(* CoDeSys 2.3.9.13 project: Stepper_03_Example01.pro *)
(* Libraries: D:\Daten\CodeSys_841\Projekte\Stepper\MC3\Release0.9.6\Stepper_03.lib 7.10.09 08:41:07, Standard.lib 22.11.04 11:21:12 *)

(* PLC configuration (modules and I/O channels)
Module Fieldbus Assignment [WAGO_Module] node 0, in %IB0 out %QB0 {INTTypePAAssignment = PLC; INTTypeModule = plugged}
Module Fieldbus Assignment [WAGO_Module] node 1, in %IB1 out %QB1 {INTTypePAAssignment = PLC; INTTypeModule = plugged}
Fieldbus variables [FB_VARS] node 1, in %IB0 out %QB0
*)

(* POU PLC_PRG, FBD *)
PROGRAM PLC_PRG
VAR
	Stepper_673					: MC3_StepperCommunication;
	Stepper1						: MC3_StepperVisu:=(	BasicModule:=673);

	Stepper1In 	AT%IB0		: ARRAY[0..11] OF BYTE;		(* input address stepper modul 750-673 *)
	Stepper1Out  	AT%QB0 		: ARRAY[0..11] OF BYTE;		(* output address stepper modul 750-673 *)


	startablauf						: BOOL;
	ablaufstate					: INT;
	error							: BOOL;
	count							: INT;
	testcount						: INT;
	TON1							: TON;
END_VAR
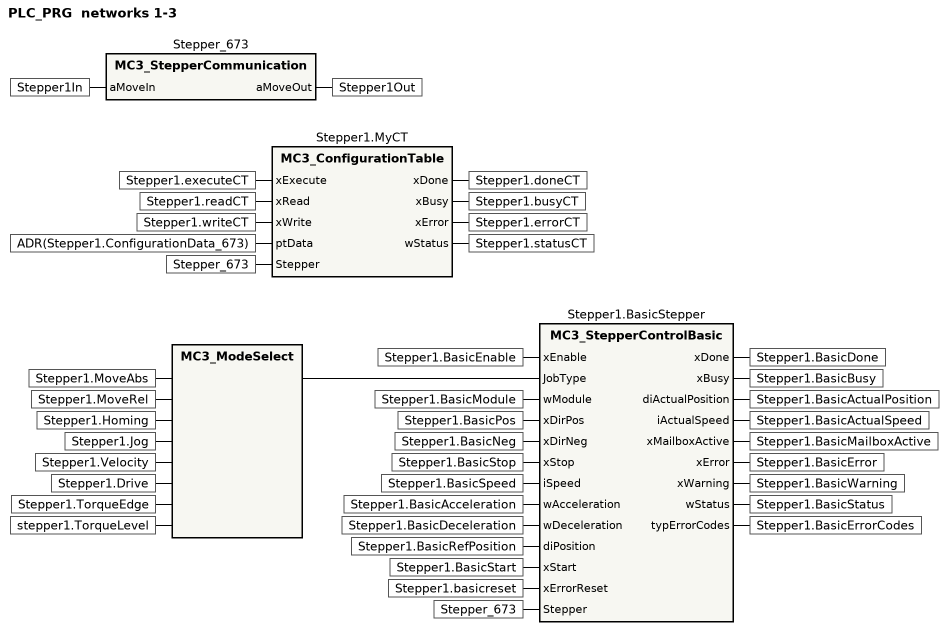
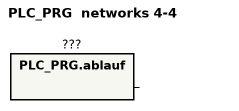
_FBD_ (* Function Block Diagram *)
NETWORK 1
	Stepper_673:MC3_StepperCommunication(aMoveIn: Stepper1In) => Stepper1Out
NETWORK 2
	Stepper1.MyCT:MC3_ConfigurationTable(xExecute: Stepper1.executeCT, xRead: Stepper1.readCT, xWrite: Stepper1.writeCT, ptData: ADR(Stepper1.ConfigurationData_673), Stepper: Stepper_673, xBusy => Stepper1.busyCT, xError => Stepper1.errorCT, wStatus => Stepper1.statusCT) => Stepper1.doneCT
NETWORK 3
	Stepper1.BasicStepper:MC3_StepperControlBasic(xEnable: Stepper1.BasicEnable, JobType: MC3_ModeSelect(Stepper1.MoveAbs, Stepper1.MoveRel, Stepper1.Homing, Stepper1.Jog, Stepper1.Velocity, Stepper1.Drive, Stepper1.TorqueEdge, stepper1.TorqueLevel), wModule: Stepper1.BasicModule, xDirPos: Stepper1.BasicPos, xDirNeg: Stepper1.BasicNeg, xStop: Stepper1.BasicStop, iSpeed: Stepper1.BasicSpeed, wAcceleration: Stepper1.BasicAcceleration, wDeceleration: Stepper1.BasicDeceleration, diPosition: Stepper1.BasicRefPosition, xStart: Stepper1.BasicStart, xErrorReset: Stepper1.basicreset, Stepper: Stepper_673, xBusy => Stepper1.BasicBusy, diActualPosition => Stepper1.BasicActualPosition, iActualSpeed => Stepper1.BasicActualSpeed, xMailboxActive => Stepper1.BasicMailboxActive, xError => Stepper1.BasicError, xWarning => Stepper1.BasicWarning, wStatus => Stepper1.BasicStatus, typErrorCodes => Stepper1.BasicErrorCodes) => Stepper1.BasicDone
NETWORK 4
	???:PLC_PRG.ablauf()
_END_FBD_
(* the same logic as Structured Text *)
(* Network 1 *)
Stepper_673(aMoveIn := Stepper1In);
Stepper1Out := Stepper_673.aMoveOut;
(* Network 2 *)
Stepper1.MyCT(xExecute := Stepper1.executeCT, xRead := Stepper1.readCT, xWrite := Stepper1.writeCT, ptData := ADR(Stepper1.ConfigurationData_673), Stepper := Stepper_673);
Stepper1.busyCT := Stepper1.MyCT.xBusy;
Stepper1.errorCT := Stepper1.MyCT.xError;
Stepper1.statusCT := Stepper1.MyCT.wStatus;
Stepper1.doneCT := Stepper1.MyCT.xDone;
(* Network 3 *)
Stepper1.BasicStepper(xEnable := Stepper1.BasicEnable, JobType := MC3_ModeSelect(Stepper1.MoveAbs, Stepper1.MoveRel, Stepper1.Homing, Stepper1.Jog, Stepper1.Velocity, Stepper1.Drive, Stepper1.TorqueEdge, stepper1.TorqueLevel), wModule := Stepper1.BasicModule, xDirPos := Stepper1.BasicPos, xDirNeg := Stepper1.BasicNeg, xStop := Stepper1.BasicStop, iSpeed := Stepper1.BasicSpeed, wAcceleration := Stepper1.BasicAcceleration, wDeceleration := Stepper1.BasicDeceleration, diPosition := Stepper1.BasicRefPosition, xStart := Stepper1.BasicStart, xErrorReset := Stepper1.basicreset, Stepper := Stepper_673);
Stepper1.BasicBusy := Stepper1.BasicStepper.xBusy;
Stepper1.BasicActualPosition := Stepper1.BasicStepper.diActualPosition;
Stepper1.BasicActualSpeed := Stepper1.BasicStepper.iActualSpeed;
Stepper1.BasicMailboxActive := Stepper1.BasicStepper.xMailboxActive;
Stepper1.BasicError := Stepper1.BasicStepper.xError;
Stepper1.BasicWarning := Stepper1.BasicStepper.xWarning;
Stepper1.BasicStatus := Stepper1.BasicStepper.wStatus;
Stepper1.BasicErrorCodes := Stepper1.BasicStepper.typErrorCodes;
Stepper1.BasicDone := Stepper1.BasicStepper.xDone;
(* Network 4: see the listing above *)
END_PROGRAM
ACTION ablauf:
IF startablauf THEN
	CASE ablaufstate OF
	0:
		Stepper1.BasicStop:=FALSE;
		Stepper1.MoveABS:=FALSE;
		Stepper1.MoveRel:=FALSE;
		Stepper1.Velocity:=FALSE;
		Stepper1.Homing:=TRUE;
		Stepper1.BasicEnable:=TRUE;
		Stepper1.BasicPos:=TRUE;
		Stepper1.BasicStart:=TRUE;
	       ablaufstate:=1;

	1:
		IF Stepper1.BasicDone THEN
      			 ablaufstate:=4;
			Stepper1.BasicPos:=FALSE;
		END_IF
	4:
		Stepper1.BasicStop:=FALSE;
		Stepper1.MoveABS:=TRUE;
		Stepper1.MoveRel:=FALSE;
		Stepper1.Velocity:=FALSE;
		Stepper1.Homing:=FALSE;
		Stepper1.BasicEnable:=TRUE;
		IF Stepper1.BasicModule=670 THEN
			Stepper1.BasicSpeed:=8000;
		ELSE
			Stepper1.BasicSpeed:=2000;
		END_IF
		Stepper1.BasicAcceleration:=1000;
		Stepper1.BasicRefPosition:=39000;
		Stepper1.BasicStart:=TRUE;

		error:=FALSE;
		ablaufstate:=5;


	5:
		IF Stepper1.BasicDone AND Stepper1.BasicStart=FALSE THEN
			Stepper1.BasicSpeed:=1500;
			Stepper1.BasicAcceleration:=1000;
			Stepper1.BasicRefPosition:=0;
			Stepper1.BasicStart:=TRUE;
			ablaufstate:=10;
		END_IF

	10:
		IF Stepper1.BasicDone THEN
			IF count>testcount THEN
				count:=0;
				IF ABS(Stepper1.BasicActualPosition)<16 THEN
					ablaufstate:=20;
				ELSE
					startablauf:=FALSE;
					error:=TRUE;
					startablauf:=FALSE;
				END_IF
			ELSE
				count:=count+1;
				ablaufstate:=4;
			END_IF
		END_IF
	20:
		Stepper1.MoveABS:=FALSE;
		Stepper1.MoveRel:=TRUE;
		Stepper1.BasicEnable:=TRUE;
		Stepper1.BasicSpeed:=4000;
		Stepper1.BasicAcceleration:=1000;
		Stepper1.BasicRefPosition:=10000;
		Stepper1.BasicStart:=TRUE;
		ablaufstate:=25;

	25:
		IF Stepper1.BasicDone THEN
			IF count>testcount THEN
				count:=0;
				ablaufstate:=30;
			ELSE
				count:=count+1;
				ablaufstate:=20;
			END_IF
		END_IF
	30:
		Stepper1.MoveABS:=FALSE;
		Stepper1.MoveRel:=FALSE;
		Stepper1.Velocity:=TRUE;
		Stepper1.BasicEnable:=TRUE;
		Stepper1.BasicSpeed:=-3000;
		Stepper1.BasicAcceleration:=300;
		Stepper1.BasicRefPosition:=10000;
		Stepper1.BasicStart:=TRUE;
		ablaufstate:=35;
	35:
		TON1(IN:=TRUE , PT:=t#5s);
		IF ton1.Q THEN
			Stepper1.BasicStop:=TRUE;
			TON1(IN:=FALSE);
			ablaufstate:=40;
		END_IF
	40:
		IF Stepper1.BasicDone THEN
			startablauf:=FALSE;
			ablaufstate:=0;
			Stepper1.BasicEnable:=FALSE;
		END_IF

	END_CASE
END_IF
END_ACTION

(* Visualisation Config763
embedded screen at (1,0)-(800,536): MC3_STEPPER_CONFIGURATION_673
*)

(* Visualisation RunStepper763
embedded screen at (0,0)-(801,538): MC3_MOVE_STEPPER_673
*)
